INTERFACE I_TraceArgument EXTENDS I_ToString

END_INTERFACE

(* stored: Version 1.1.0.1, ProductVersion 3.1.4026.18
   Itf I_TraceArgument: Id {61b1e66b-4c6d-0789-1082-50edb71ae090} *)
